// LS Electric XG5000 project: 동남135
// PLC NewPLC
// module base 0 slot 0: 입출력 모듈:XBC-DN/DP14E (DC 24V 입력 8점, 트랜지스터 출력 6점)

PROGRAM NewProgram (task: 스캔 프로그램)

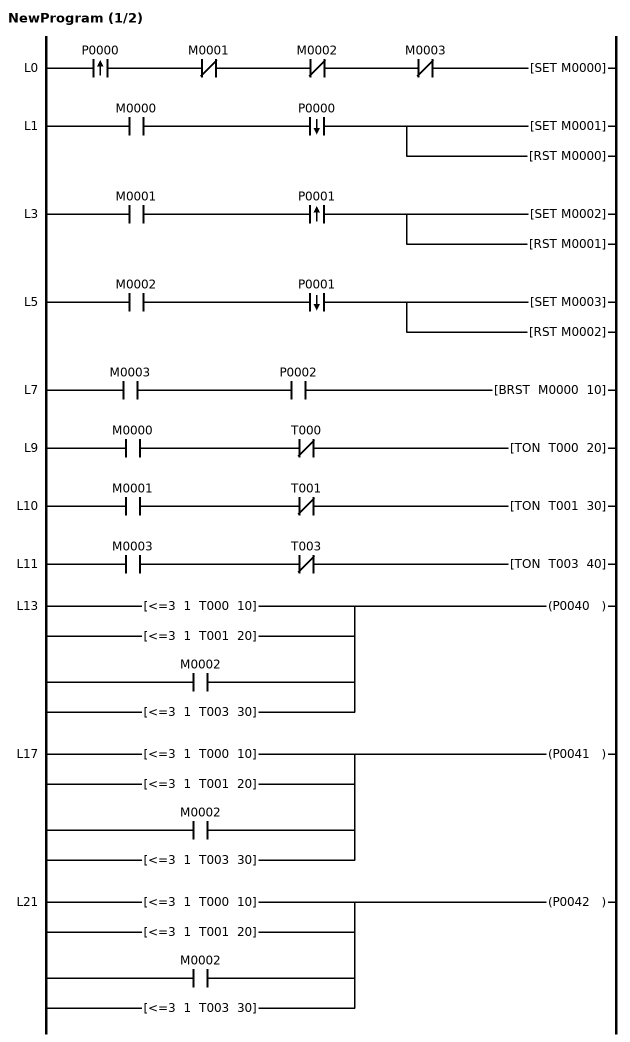
; L0
LOADP     P0000
AND NOT   M0001
AND NOT   M0002
AND NOT   M0003
SET       M0000
; L1
LOAD      M0000
ANDN      P0000
SET       M0001
RST       M0000
; L3
LOAD      M0001
ANDP      P0001
SET       M0002
RST       M0001
; L5
LOAD      M0002
ANDN      P0001
SET       M0003
RST       M0002
; L7
LOAD      M0003
AND       P0002
BRST      M0000 10
; L9
LOAD      M0000
AND NOT   T000
TON       T000 20
; L10
LOAD      M0001
AND NOT   T001
TON       T001 30
; L11
LOAD      M0003
AND NOT   T003
TON       T003 40
; L13
LOAD<=3   1 T000 10
OR<=3     1 T001 20
OR        M0002
OR<=3     1 T003 30
OUT       P0040
; L17
LOAD<=3   1 T000 10
OR<=3     1 T001 20
OR        M0002
OR<=3     1 T003 30
OUT       P0041
; L21
LOAD<=3   1 T000 10
OR<=3     1 T001 20
OR        M0002
OR<=3     1 T003 30
OUT       P0042

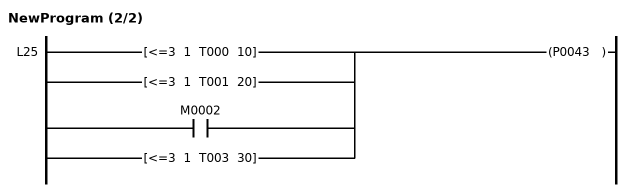
; L25
LOAD<=3   1 T000 10
OR<=3     1 T001 20
OR        M0002
OR<=3     1 T003 30
OUT       P0043